(* PLC project Unnamed, Unknown Unnamed 1 *)
(* stored: creationDateTime 2024-01-09T16:45:07, modificationDateTime 2024-01-23T14:31:54 *)

FUNCTION_BLOCK Reals_MultiplyByParameter
  VAR_INPUT
    u : REAL;
    k : REAL;
  END_VAR
  VAR_OUTPUT
    y : REAL;
  END_VAR

						y := k * u;
					
END_FUNCTION_BLOCK

PROGRAM MultiplyByParameter_1
  VAR_INPUT
    u2 : REAL;
  END_VAR
  VAR_OUTPUT
    y1 : REAL;
  END_VAR
  VAR
    gain : Reals_MultiplyByParameter;
    _1 : REAL := 1.0;
  END_VAR

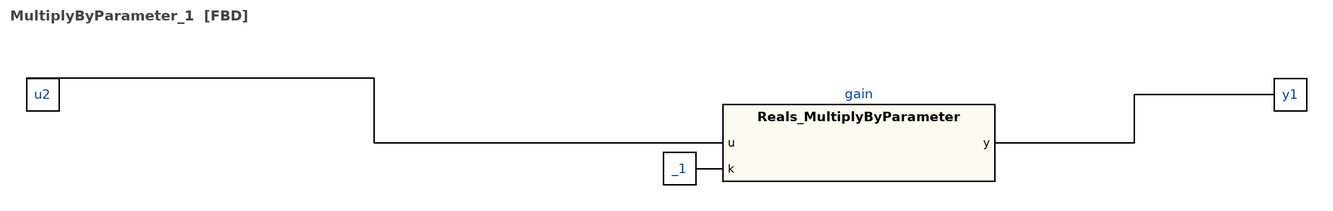
(* FBD diagram, written out as Structured Text *)
gain(u := u2, k := _1);
y1 := gain.y;
END_PROGRAM

CONFIGURATION config
  RESOURCE resource1 ON PLC
    TASK task0(INTERVAL := T#20ms, PRIORITY := 0);
    PROGRAM instance0 WITH task0 : MultiplyByParameter_1;
  END_RESOURCE
END_CONFIGURATION
